TYPE ST_SlaveJointData :
STRUCT
	
	// joint position compute with motor encoder
	m_curMotorPos :ARRAY[1..g_sArmNum, 1..g_sJntNum] OF LREAL;
	
	// joint position compute with link/abs encoder
	m_curLinkPos :ARRAY[1..g_sArmNum, 1..g_sJntNum] OF LREAL;
	
	// target joint position 
	m_cmdJntPos :ARRAY[1..g_sArmNum, 1..g_sJntNum] OF LREAL;
	
	// current joint position 
	m_curJntPos :ARRAY[1..g_sArmNum, 1..g_sJntNum] OF LREAL;
	
	// target joint velocity 
	m_cmdJntVel :ARRAY[1..g_sArmNum, 1..g_sJntNum] OF LREAL;
	
	// current joint position 
	m_curJntVel :ARRAY[1..g_sArmNum, 1..g_sJntNum] OF LREAL;
	
	// command joint torque 
	m_cmdJntTrq :ARRAY[1..g_sArmNum, 1..g_sJntNum] OF LREAL;
	
	// current joint torque 
	m_curJntTrq :ARRAY[1..g_sArmNum, 1..g_sJntNum] OF LREAL;
END_STRUCT
END_TYPE

(* stored: Version 1.1.0.1, ProductVersion 3.1.4024.12
   DUT ST_SlaveJointData: Id {775e1618-4069-46ed-920d-0e7ed2d13e2f} *)
